FUNCTION_BLOCK A2X2_4AX_TO_2X (* Composite FB for convert 4 AX to A2X2 *)
  (* Standard: 61499-2; Function: A2X2 has 2 channels (UP/DOWN), each bidirectional, so it takes 4 unidirectional AX to represent it: IND_UP/IND_DOWN carry what gets published by A2X2_OUT (its EO_UP/EO_DOWN indication side), REQ_UP/REQ_DOWN carry what A2X2_OUT receives back (its EI_UP/EI_DOWN request side).; Description: Copyright (c) 2026 HR Agrartechnik GmbH This program and the accompanying materials are made available under the terms of the Eclipse Public License 2.0 which is available at https://www.eclipse.org/legal/epl-2.0/ SPDX-License-Identifier: EPL-2.0 *)
  (* Version 1.0, 2026-08-31, Franz Höpfinger, HR Agrartechnik GmbH, Initial Version *)
  PACKAGE adapter::conversion::bidirectional;
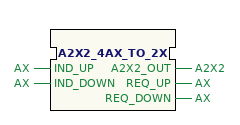
  SOCKETS
    IND_UP : adapter::types::unidirectional::AX; (* Indication UP, received from outside, forwarded into A2X2_OUT.EO_UP *)
    IND_DOWN : adapter::types::unidirectional::AX; (* Indication DOWN, received from outside, forwarded into A2X2_OUT.EO_DOWN *)
  END_SOCKETS
  PLUGS
    A2X2_OUT : adapter::types::bidirectional::A2X2; (* Adapter Output *)
    REQ_UP : adapter::types::unidirectional::AX; (* Request UP, published outward from A2X2_OUT.EI_UP *)
    REQ_DOWN : adapter::types::unidirectional::AX; (* Request DOWN, published outward from A2X2_OUT.EI_DOWN *)
  END_PLUGS
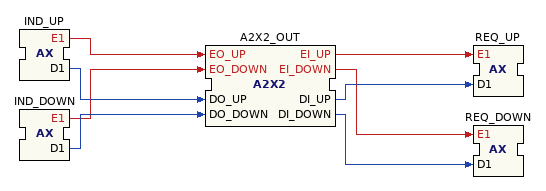
  EVENT_CONNECTIONS
    IND_UP.E1 TO A2X2_OUT.EO_UP;
    IND_DOWN.E1 TO A2X2_OUT.EO_DOWN;
    A2X2_OUT.EI_UP TO REQ_UP.E1;
    A2X2_OUT.EI_DOWN TO REQ_DOWN.E1;
  END_CONNECTIONS
  DATA_CONNECTIONS
    IND_UP.D1 TO A2X2_OUT.DO_UP;
    IND_DOWN.D1 TO A2X2_OUT.DO_DOWN;
    A2X2_OUT.DI_UP TO REQ_UP.D1;
    A2X2_OUT.DI_DOWN TO REQ_DOWN.D1;
  END_CONNECTIONS
END_FUNCTION_BLOCK
